FUNCTION_BLOCK PAMMixer EXTENDS PAProcessModule
VAR_INPUT
END_VAR
VAR_OUTPUT
END_VAR
VAR
	_PAPointMatIn1 : PAPoint(THIS^);
	_PAPointMatOut1 : PAPoint(THIS^);
END_VAR

METHOD FB_init : BOOL
VAR_INPUT
	bInitRetains : BOOL; // if TRUE, the retain variables are initialized (warm start / cold start)
	bInCopyCode : BOOL;  // if TRUE, the instance afterwards gets moved into the copy code (online change)
	parent : IACComponent;
END_VAR
AddPoint(_PAPointMatIn1);
AddPoint(_PAPointMatOut1);
END_METHOD

PROPERTY PUBLIC PAPointMatIn1 : IACPoint
GET
PAPointMatIn1 := _PAPointMatIn1;
END_GET
END_PROPERTY

PROPERTY PUBLIC PAPointMatOut1 : IACPoint
GET
PAPointMatOut1 := _PAPointMatOut1;
END_GET
END_PROPERTY

END_FUNCTION_BLOCK

(* stored: Version 1.1.0.1, ProductVersion 3.1.4020.12
   POU PAMMixer: Id {ee264b77-81b1-4f2c-a22e-035c761b8925}, SpecialFunc None
   Method FB_init: Id {28759f57-1141-4b94-ac42-da86149e36db}
   Property PAPointMatIn1: Id {069dec9c-64d6-4962-894f-df591da53eac}
   Get Get: Id {8b944920-b037-40e7-94e4-e0efe80bbe9e}
   Property PAPointMatOut1: Id {e7ec3235-dcd4-4bcc-935b-57b513d1e506}
   Get Get: Id {9b26c0db-f75a-4320-aa36-e2b657b418da} *)
